(* PLC project SyntheticProject, CODESYS CODESYS V3.5 SP21 *)
(* stored: creationDateTime 2026-07-17T11:48:53, modificationDateTime 2026-07-17T11:48:53 *)

TYPE E_StationMode : (IDLE := 0, ACQUIRE := 10);
END_TYPE

TYPE E_MachineState : (OFF := 0);
END_TYPE

{attribute 'qualified_only'}
TYPE E_AlarmClass : (None := 0);
END_TYPE

TYPE ST_AxisConfig : STRUCT
  rMaxVel : REAL;  (* Max velocity *)
  rMaxAcc : REAL;  (* Max acceleration *)
  rMaxDec : REAL;  (* Max deceleration *)
  nAxisId : INT;  (* Axis identifier *)
  bInverted : BOOL;  (* Direction inverted *)
  tTimeout : TIME;  (* Motion timeout *)
END_STRUCT;
END_TYPE

TYPE ST_StationStats : STRUCT
  nTotalCycles : UDINT;  (* Total cycles run *)
  nFaultCount : DINT;  (* Fault count *)
  lrUptimeSec : LREAL;  (* Uptime in seconds *)
  rLastPos : REAL;  (* Last actual position *)
  sLastFault : STRING;  (* Last fault text *)
END_STRUCT;
END_TYPE

VAR_GLOBAL  (* GVL_Machine *)
  bMachineReady : BOOL;  (* Machine ready flag *)
  bEStop : BOOL;  (* Emergency stop active *)
  eMachineMode : E_MachineState;  (* Current machine state *)
  stAxisCfg : ST_AxisConfig;  (* Shared axis config *)
  nActiveStation : INT := 0;  (* Active station index *)
  rLineSpeed : REAL := 0.0;  (* Line speed *)
  lrProduced : LREAL := 0.0;  (* Produced count (long) *)
  tHeartbeat : TIME;  (* Heartbeat period *)
  sMachineName : STRING := 'LineA';  (* Machine name *)
END_VAR

VAR_GLOBAL CONSTANT  (* GVL_Config *)
  nMaxStations : INT := 24;  (* Max stations *)
  nBufferSize : UDINT := 256;  (* Buffer size *)
  rPi : REAL := 3.14159;  (* Pi constant *)
  lrGravity : LREAL := 9.80665;  (* Gravity constant *)
  tCycleTimeout : TIME := T#5S;  (* Default cycle timeout *)
  sVersion : STRING := '1.0.0';  (* Fixture version *)
END_VAR

VAR_GLOBAL RETAIN PERSISTENT  (* GVL_Persist *)
  nPowerCycles : UDINT := 0;  (* Power-cycle counter *)
  rTotalRuntime : LREAL := 0.0;  (* Accumulated runtime [h] *)
  nLastRecipeId : INT := 0;  (* Recipe restored on boot *)
END_VAR

FUNCTION_BLOCK FB_Debounce
  VAR_INPUT
    bIn : BOOL;  (* Raw input *)
    tDebounce : TIME := T#20MS;  (* Debounce time *)
  END_VAR
  VAR_OUTPUT
    bOut : BOOL;  (* Debounced output *)
  END_VAR
  VAR
    nState : INT := 0;  (* State machine *)
    bLast : BOOL;  (* Last raw sample *)
  END_VAR

          CASE nState OF
    0: // IDLE
        IF bIn <> bLast THEN
            nState := 10;
        END_IF
    10: // SETTLING
        bLast := bIn;
        bOut := bIn;
        nState := 0;
END_CASE
        
END_FUNCTION_BLOCK

FUNCTION_BLOCK FB_Delay
  VAR_INPUT
    bStart : BOOL;  (* Start the delay *)
    tDelay : TIME := T#1S;  (* Delay duration *)
  END_VAR
  VAR_OUTPUT
    bDone : BOOL;  (* Delay elapsed *)
  END_VAR
  VAR
    nState : INT := 0;  (* State machine *)
    tElapsed : TIME;  (* Accumulated time *)
  END_VAR

          CASE nState OF
    0: // IDLE
        bDone := FALSE;
        IF bStart THEN
            nState := 10;
        END_IF
    10: // TIMING
        bDone := TRUE;
        nState := 90;
    90: // DONE
        IF NOT bStart THEN
            nState := 0;
        END_IF
END_CASE
        
END_FUNCTION_BLOCK

FUNCTION_BLOCK FB_Station01
  VAR_INPUT
    bEnable : BOOL;  (* Enable this station *)
    bExecute : BOOL;  (* Trigger one work cycle *)
    bReset : BOOL;  (* Clear latched error *)
    nMode : INT := 0;  (* Operating mode selector *)
    rSetpoint : REAL := 0.0;  (* Target setpoint *)
    tTimeout : TIME := T#5S;  (* Watchdog timeout *)
    sLabel : STRING := 'station';  (* Human-readable label *)
    nStationId : DINT := 1;  (* Station identifier *)
  END_VAR
  VAR_OUTPUT
    bDone : BOOL;  (* Cycle finished *)
    bBusy : BOOL;  (* Cycle running *)
    bErr : BOOL;  (* Error latched *)
    nErrId : DINT := 0;  (* Active error code *)
    rActPos : REAL;  (* Actual position feedback *)
    nCycleCount : UDINT := 0;  (* Completed cycle counter *)
  END_VAR
  VAR
    nState : INT := 0;  (* State machine register *)
    fbSub : FB_Debounce;  (* Nested FB instance *)
    fbTimer : FB_Delay;  (* Nested FB instance *)
    anBuffer : ARRAY[0..9] OF INT;  (* Integer ring buffer *)
    arSamples : ARRAY[0..7] OF REAL;  (* Sample window *)
    lrAccum : LREAL := 0.0;  (* Long accumulator *)
    tElapsed : TIME;  (* Elapsed cycle time *)
    bInternal : BOOL;  (* Internal work flag *)
  END_VAR
  VAR CONSTANT
    nMaxRetries : INT := 3;  (* Retry limit *)
    rScale : REAL := 1.5;  (* Setpoint scale factor *)
  END_VAR

          // 01: main state machine — 0 IDLE / 10-20 WORK / 90 DONE / 99 ERROR
CASE nState OF
    0: // IDLE — wait for enable + execute
        bBusy := FALSE;
        bDone := FALSE;
        IF bEnable AND bExecute THEN
            nState := 10;
        END_IF

    10: // WORK: acquire
        bBusy := TRUE;
        nCycleCount := nCycleCount + 1;
        fbSub(bIn := bEnable);
        nState := 20;

    20: (* WORK: process the sample and compute position *)
        rActPos := rSetpoint * rScale;
        lrAccum := lrAccum + LREAL#TO_LREAL(rActPos);
        fbTimer(bStart := TRUE, tDelay := tTimeout);
        IF fbTimer.bDone THEN
            nState := 90;
        END_IF

    90: // DONE — publish result, return to idle
        bDone := TRUE;
        bBusy := FALSE;
        nState := 0;

    99: // ERROR — latch fault
        bErr := TRUE;
        nErrId := 16#8001;
        bBusy := FALSE;
END_CASE

// Global reset path
IF bReset THEN
    bErr := FALSE;
    nErrId := 0;
    nState := 0;
END_IF
        
END_FUNCTION_BLOCK

FUNCTION_BLOCK FB_Station02
  VAR_INPUT
    bEnable : BOOL;  (* Enable this station *)
    bExecute : BOOL;  (* Trigger one work cycle *)
    bReset : BOOL;  (* Clear latched error *)
    nMode : INT := 0;  (* Operating mode selector *)
    rSetpoint : REAL := 0.0;  (* Target setpoint *)
    tTimeout : TIME := T#5S;  (* Watchdog timeout *)
    sLabel : STRING := 'station';  (* Human-readable label *)
    nStationId : DINT := 2;  (* Station identifier *)
  END_VAR
  VAR_OUTPUT
    bDone : BOOL;  (* Cycle finished *)
    bBusy : BOOL;  (* Cycle running *)
    bErr : BOOL;  (* Error latched *)
    nErrId : DINT := 0;  (* Active error code *)
    rActPos : REAL;  (* Actual position feedback *)
    nCycleCount : UDINT := 0;  (* Completed cycle counter *)
  END_VAR
  VAR
    nState : INT := 0;  (* State machine register *)
    fbSub : FB_Debounce;  (* Nested FB instance *)
    fbTimer : FB_Delay;  (* Nested FB instance *)
    anBuffer : ARRAY[0..9] OF INT;  (* Integer ring buffer *)
    arSamples : ARRAY[0..7] OF REAL;  (* Sample window *)
    lrAccum : LREAL := 0.0;  (* Long accumulator *)
    tElapsed : TIME;  (* Elapsed cycle time *)
    bInternal : BOOL;  (* Internal work flag *)
  END_VAR
  VAR CONSTANT
    nMaxRetries : INT := 3;  (* Retry limit *)
    rScale : REAL := 1.5;  (* Setpoint scale factor *)
  END_VAR

          // 02: main state machine — 0 IDLE / 10-20 WORK / 90 DONE / 99 ERROR
CASE nState OF
    0: // IDLE — wait for enable + execute
        bBusy := FALSE;
        bDone := FALSE;
        IF bEnable AND bExecute THEN
            nState := 10;
        END_IF

    10: // WORK: acquire
        bBusy := TRUE;
        nCycleCount := nCycleCount + 1;
        fbSub(bIn := bEnable);
        nState := 20;

    20: (* WORK: process the sample and compute position *)
        rActPos := rSetpoint * rScale;
        lrAccum := lrAccum + LREAL#TO_LREAL(rActPos);
        fbTimer(bStart := TRUE, tDelay := tTimeout);
        IF fbTimer.bDone THEN
            nState := 90;
        END_IF

    90: // DONE — publish result, return to idle
        bDone := TRUE;
        bBusy := FALSE;
        nState := 0;

    99: // ERROR — latch fault
        bErr := TRUE;
        nErrId := 16#8001;
        bBusy := FALSE;
END_CASE

// Global reset path
IF bReset THEN
    bErr := FALSE;
    nErrId := 0;
    nState := 0;
END_IF
        
END_FUNCTION_BLOCK

FUNCTION_BLOCK FB_Station03
  VAR_INPUT
    bEnable : BOOL;  (* Enable this station *)
    bExecute : BOOL;  (* Trigger one work cycle *)
    bReset : BOOL;  (* Clear latched error *)
    nMode : INT := 0;  (* Operating mode selector *)
    rSetpoint : REAL := 0.0;  (* Target setpoint *)
    tTimeout : TIME := T#5S;  (* Watchdog timeout *)
    sLabel : STRING := 'station';  (* Human-readable label *)
    nStationId : DINT := 3;  (* Station identifier *)
  END_VAR
  VAR_OUTPUT
    bDone : BOOL;  (* Cycle finished *)
    bBusy : BOOL;  (* Cycle running *)
    bErr : BOOL;  (* Error latched *)
    nErrId : DINT := 0;  (* Active error code *)
    rActPos : REAL;  (* Actual position feedback *)
    nCycleCount : UDINT := 0;  (* Completed cycle counter *)
  END_VAR
  VAR
    nState : INT := 0;  (* State machine register *)
    fbSub : FB_Debounce;  (* Nested FB instance *)
    fbTimer : FB_Delay;  (* Nested FB instance *)
    anBuffer : ARRAY[0..9] OF INT;  (* Integer ring buffer *)
    arSamples : ARRAY[0..7] OF REAL;  (* Sample window *)
    lrAccum : LREAL := 0.0;  (* Long accumulator *)
    tElapsed : TIME;  (* Elapsed cycle time *)
    bInternal : BOOL;  (* Internal work flag *)
  END_VAR
  VAR CONSTANT
    nMaxRetries : INT := 3;  (* Retry limit *)
    rScale : REAL := 1.5;  (* Setpoint scale factor *)
  END_VAR

          // 03: main state machine — 0 IDLE / 10-20 WORK / 90 DONE / 99 ERROR
CASE nState OF
    0: // IDLE — wait for enable + execute
        bBusy := FALSE;
        bDone := FALSE;
        IF bEnable AND bExecute THEN
            nState := 10;
        END_IF

    10: // WORK: acquire
        bBusy := TRUE;
        nCycleCount := nCycleCount + 1;
        fbSub(bIn := bEnable);
        nState := 20;

    20: (* WORK: process the sample and compute position *)
        rActPos := rSetpoint * rScale;
        lrAccum := lrAccum + LREAL#TO_LREAL(rActPos);
        fbTimer(bStart := TRUE, tDelay := tTimeout);
        IF fbTimer.bDone THEN
            nState := 90;
        END_IF

    90: // DONE — publish result, return to idle
        bDone := TRUE;
        bBusy := FALSE;
        nState := 0;

    99: // ERROR — latch fault
        bErr := TRUE;
        nErrId := 16#8001;
        bBusy := FALSE;
END_CASE

// Global reset path
IF bReset THEN
    bErr := FALSE;
    nErrId := 0;
    nState := 0;
END_IF
        
END_FUNCTION_BLOCK

FUNCTION_BLOCK FB_Station04
  VAR_INPUT
    bEnable : BOOL;  (* Enable this station *)
    bExecute : BOOL;  (* Trigger one work cycle *)
    bReset : BOOL;  (* Clear latched error *)
    nMode : INT := 0;  (* Operating mode selector *)
    rSetpoint : REAL := 0.0;  (* Target setpoint *)
    tTimeout : TIME := T#5S;  (* Watchdog timeout *)
    sLabel : STRING := 'station';  (* Human-readable label *)
    nStationId : DINT := 4;  (* Station identifier *)
  END_VAR
  VAR_OUTPUT
    bDone : BOOL;  (* Cycle finished *)
    bBusy : BOOL;  (* Cycle running *)
    bErr : BOOL;  (* Error latched *)
    nErrId : DINT := 0;  (* Active error code *)
    rActPos : REAL;  (* Actual position feedback *)
    nCycleCount : UDINT := 0;  (* Completed cycle counter *)
  END_VAR
  VAR
    nState : INT := 0;  (* State machine register *)
    fbSub : FB_Debounce;  (* Nested FB instance *)
    fbTimer : FB_Delay;  (* Nested FB instance *)
    anBuffer : ARRAY[0..9] OF INT;  (* Integer ring buffer *)
    arSamples : ARRAY[0..7] OF REAL;  (* Sample window *)
    lrAccum : LREAL := 0.0;  (* Long accumulator *)
    tElapsed : TIME;  (* Elapsed cycle time *)
    bInternal : BOOL;  (* Internal work flag *)
  END_VAR
  VAR CONSTANT
    nMaxRetries : INT := 3;  (* Retry limit *)
    rScale : REAL := 1.5;  (* Setpoint scale factor *)
  END_VAR

          // 04: main state machine — 0 IDLE / 10-20 WORK / 90 DONE / 99 ERROR
CASE nState OF
    0: // IDLE — wait for enable + execute
        bBusy := FALSE;
        bDone := FALSE;
        IF bEnable AND bExecute THEN
            nState := 10;
        END_IF

    10: // WORK: acquire
        bBusy := TRUE;
        nCycleCount := nCycleCount + 1;
        fbSub(bIn := bEnable);
        nState := 20;

    20: (* WORK: process the sample and compute position *)
        rActPos := rSetpoint * rScale;
        lrAccum := lrAccum + LREAL#TO_LREAL(rActPos);
        fbTimer(bStart := TRUE, tDelay := tTimeout);
        IF fbTimer.bDone THEN
            nState := 90;
        END_IF

    90: // DONE — publish result, return to idle
        bDone := TRUE;
        bBusy := FALSE;
        nState := 0;

    99: // ERROR — latch fault
        bErr := TRUE;
        nErrId := 16#8001;
        bBusy := FALSE;
END_CASE

// Global reset path
IF bReset THEN
    bErr := FALSE;
    nErrId := 0;
    nState := 0;
END_IF
        
END_FUNCTION_BLOCK

FUNCTION_BLOCK FB_Station05
  VAR_INPUT
    bEnable : BOOL;  (* Enable this station *)
    bExecute : BOOL;  (* Trigger one work cycle *)
    bReset : BOOL;  (* Clear latched error *)
    nMode : INT := 0;  (* Operating mode selector *)
    rSetpoint : REAL := 0.0;  (* Target setpoint *)
    tTimeout : TIME := T#5S;  (* Watchdog timeout *)
    sLabel : STRING := 'station';  (* Human-readable label *)
    nStationId : DINT := 5;  (* Station identifier *)
  END_VAR
  VAR_OUTPUT
    bDone : BOOL;  (* Cycle finished *)
    bBusy : BOOL;  (* Cycle running *)
    bErr : BOOL;  (* Error latched *)
    nErrId : DINT := 0;  (* Active error code *)
    rActPos : REAL;  (* Actual position feedback *)
    nCycleCount : UDINT := 0;  (* Completed cycle counter *)
  END_VAR
  VAR
    nState : INT := 0;  (* State machine register *)
    fbSub : FB_Debounce;  (* Nested FB instance *)
    fbTimer : FB_Delay;  (* Nested FB instance *)
    anBuffer : ARRAY[0..9] OF INT;  (* Integer ring buffer *)
    arSamples : ARRAY[0..7] OF REAL;  (* Sample window *)
    lrAccum : LREAL := 0.0;  (* Long accumulator *)
    tElapsed : TIME;  (* Elapsed cycle time *)
    bInternal : BOOL;  (* Internal work flag *)
  END_VAR
  VAR CONSTANT
    nMaxRetries : INT := 3;  (* Retry limit *)
    rScale : REAL := 1.5;  (* Setpoint scale factor *)
  END_VAR

          // 05: main state machine — 0 IDLE / 10-20 WORK / 90 DONE / 99 ERROR
CASE nState OF
    0: // IDLE — wait for enable + execute
        bBusy := FALSE;
        bDone := FALSE;
        IF bEnable AND bExecute THEN
            nState := 10;
        END_IF

    10: // WORK: acquire
        bBusy := TRUE;
        nCycleCount := nCycleCount + 1;
        fbSub(bIn := bEnable);
        nState := 20;

    20: (* WORK: process the sample and compute position *)
        rActPos := rSetpoint * rScale;
        lrAccum := lrAccum + LREAL#TO_LREAL(rActPos);
        fbTimer(bStart := TRUE, tDelay := tTimeout);
        IF fbTimer.bDone THEN
            nState := 90;
        END_IF

    90: // DONE — publish result, return to idle
        bDone := TRUE;
        bBusy := FALSE;
        nState := 0;

    99: // ERROR — latch fault
        bErr := TRUE;
        nErrId := 16#8001;
        bBusy := FALSE;
END_CASE

// Global reset path
IF bReset THEN
    bErr := FALSE;
    nErrId := 0;
    nState := 0;
END_IF
        
END_FUNCTION_BLOCK

FUNCTION_BLOCK FB_Station06
  VAR_INPUT
    bEnable : BOOL;  (* Enable this station *)
    bExecute : BOOL;  (* Trigger one work cycle *)
    bReset : BOOL;  (* Clear latched error *)
    nMode : INT := 0;  (* Operating mode selector *)
    rSetpoint : REAL := 0.0;  (* Target setpoint *)
    tTimeout : TIME := T#5S;  (* Watchdog timeout *)
    sLabel : STRING := 'station';  (* Human-readable label *)
    nStationId : DINT := 6;  (* Station identifier *)
  END_VAR
  VAR_OUTPUT
    bDone : BOOL;  (* Cycle finished *)
    bBusy : BOOL;  (* Cycle running *)
    bErr : BOOL;  (* Error latched *)
    nErrId : DINT := 0;  (* Active error code *)
    rActPos : REAL;  (* Actual position feedback *)
    nCycleCount : UDINT := 0;  (* Completed cycle counter *)
  END_VAR
  VAR
    nState : INT := 0;  (* State machine register *)
    fbSub : FB_Debounce;  (* Nested FB instance *)
    fbTimer : FB_Delay;  (* Nested FB instance *)
    anBuffer : ARRAY[0..9] OF INT;  (* Integer ring buffer *)
    arSamples : ARRAY[0..7] OF REAL;  (* Sample window *)
    lrAccum : LREAL := 0.0;  (* Long accumulator *)
    tElapsed : TIME;  (* Elapsed cycle time *)
    bInternal : BOOL;  (* Internal work flag *)
  END_VAR
  VAR CONSTANT
    nMaxRetries : INT := 3;  (* Retry limit *)
    rScale : REAL := 1.5;  (* Setpoint scale factor *)
  END_VAR

          // 06: main state machine — 0 IDLE / 10-20 WORK / 90 DONE / 99 ERROR
CASE nState OF
    0: // IDLE — wait for enable + execute
        bBusy := FALSE;
        bDone := FALSE;
        IF bEnable AND bExecute THEN
            nState := 10;
        END_IF

    10: // WORK: acquire
        bBusy := TRUE;
        nCycleCount := nCycleCount + 1;
        fbSub(bIn := bEnable);
        nState := 20;

    20: (* WORK: process the sample and compute position *)
        rActPos := rSetpoint * rScale;
        lrAccum := lrAccum + LREAL#TO_LREAL(rActPos);
        fbTimer(bStart := TRUE, tDelay := tTimeout);
        IF fbTimer.bDone THEN
            nState := 90;
        END_IF

    90: // DONE — publish result, return to idle
        bDone := TRUE;
        bBusy := FALSE;
        nState := 0;

    99: // ERROR — latch fault
        bErr := TRUE;
        nErrId := 16#8001;
        bBusy := FALSE;
END_CASE

// Global reset path
IF bReset THEN
    bErr := FALSE;
    nErrId := 0;
    nState := 0;
END_IF
        
END_FUNCTION_BLOCK

FUNCTION_BLOCK FB_Station07
  VAR_INPUT
    bEnable : BOOL;  (* Enable this station *)
    bExecute : BOOL;  (* Trigger one work cycle *)
    bReset : BOOL;  (* Clear latched error *)
    nMode : INT := 0;  (* Operating mode selector *)
    rSetpoint : REAL := 0.0;  (* Target setpoint *)
    tTimeout : TIME := T#5S;  (* Watchdog timeout *)
    sLabel : STRING := 'station';  (* Human-readable label *)
    nStationId : DINT := 7;  (* Station identifier *)
  END_VAR
  VAR_OUTPUT
    bDone : BOOL;  (* Cycle finished *)
    bBusy : BOOL;  (* Cycle running *)
    bErr : BOOL;  (* Error latched *)
    nErrId : DINT := 0;  (* Active error code *)
    rActPos : REAL;  (* Actual position feedback *)
    nCycleCount : UDINT := 0;  (* Completed cycle counter *)
  END_VAR
  VAR
    nState : INT := 0;  (* State machine register *)
    fbSub : FB_Debounce;  (* Nested FB instance *)
    fbTimer : FB_Delay;  (* Nested FB instance *)
    anBuffer : ARRAY[0..9] OF INT;  (* Integer ring buffer *)
    arSamples : ARRAY[0..7] OF REAL;  (* Sample window *)
    lrAccum : LREAL := 0.0;  (* Long accumulator *)
    tElapsed : TIME;  (* Elapsed cycle time *)
    bInternal : BOOL;  (* Internal work flag *)
  END_VAR
  VAR CONSTANT
    nMaxRetries : INT := 3;  (* Retry limit *)
    rScale : REAL := 1.5;  (* Setpoint scale factor *)
  END_VAR

          // 07: main state machine — 0 IDLE / 10-20 WORK / 90 DONE / 99 ERROR
CASE nState OF
    0: // IDLE — wait for enable + execute
        bBusy := FALSE;
        bDone := FALSE;
        IF bEnable AND bExecute THEN
            nState := 10;
        END_IF

    10: // WORK: acquire
        bBusy := TRUE;
        nCycleCount := nCycleCount + 1;
        fbSub(bIn := bEnable);
        nState := 20;

    20: (* WORK: process the sample and compute position *)
        rActPos := rSetpoint * rScale;
        lrAccum := lrAccum + LREAL#TO_LREAL(rActPos);
        fbTimer(bStart := TRUE, tDelay := tTimeout);
        IF fbTimer.bDone THEN
            nState := 90;
        END_IF

    90: // DONE — publish result, return to idle
        bDone := TRUE;
        bBusy := FALSE;
        nState := 0;

    99: // ERROR — latch fault
        bErr := TRUE;
        nErrId := 16#8001;
        bBusy := FALSE;
END_CASE

// Global reset path
IF bReset THEN
    bErr := FALSE;
    nErrId := 0;
    nState := 0;
END_IF
        
END_FUNCTION_BLOCK

FUNCTION_BLOCK FB_Station08
  VAR_INPUT
    bEnable : BOOL;  (* Enable this station *)
    bExecute : BOOL;  (* Trigger one work cycle *)
    bReset : BOOL;  (* Clear latched error *)
    nMode : INT := 0;  (* Operating mode selector *)
    rSetpoint : REAL := 0.0;  (* Target setpoint *)
    tTimeout : TIME := T#5S;  (* Watchdog timeout *)
    sLabel : STRING := 'station';  (* Human-readable label *)
    nStationId : DINT := 8;  (* Station identifier *)
  END_VAR
  VAR_OUTPUT
    bDone : BOOL;  (* Cycle finished *)
    bBusy : BOOL;  (* Cycle running *)
    bErr : BOOL;  (* Error latched *)
    nErrId : DINT := 0;  (* Active error code *)
    rActPos : REAL;  (* Actual position feedback *)
    nCycleCount : UDINT := 0;  (* Completed cycle counter *)
  END_VAR
  VAR
    nState : INT := 0;  (* State machine register *)
    fbSub : FB_Debounce;  (* Nested FB instance *)
    fbTimer : FB_Delay;  (* Nested FB instance *)
    anBuffer : ARRAY[0..9] OF INT;  (* Integer ring buffer *)
    arSamples : ARRAY[0..7] OF REAL;  (* Sample window *)
    lrAccum : LREAL := 0.0;  (* Long accumulator *)
    tElapsed : TIME;  (* Elapsed cycle time *)
    bInternal : BOOL;  (* Internal work flag *)
  END_VAR
  VAR CONSTANT
    nMaxRetries : INT := 3;  (* Retry limit *)
    rScale : REAL := 1.5;  (* Setpoint scale factor *)
  END_VAR

          // 08: main state machine — 0 IDLE / 10-20 WORK / 90 DONE / 99 ERROR
CASE nState OF
    0: // IDLE — wait for enable + execute
        bBusy := FALSE;
        bDone := FALSE;
        IF bEnable AND bExecute THEN
            nState := 10;
        END_IF

    10: // WORK: acquire
        bBusy := TRUE;
        nCycleCount := nCycleCount + 1;
        fbSub(bIn := bEnable);
        nState := 20;

    20: (* WORK: process the sample and compute position *)
        rActPos := rSetpoint * rScale;
        lrAccum := lrAccum + LREAL#TO_LREAL(rActPos);
        fbTimer(bStart := TRUE, tDelay := tTimeout);
        IF fbTimer.bDone THEN
            nState := 90;
        END_IF

    90: // DONE — publish result, return to idle
        bDone := TRUE;
        bBusy := FALSE;
        nState := 0;

    99: // ERROR — latch fault
        bErr := TRUE;
        nErrId := 16#8001;
        bBusy := FALSE;
END_CASE

// Global reset path
IF bReset THEN
    bErr := FALSE;
    nErrId := 0;
    nState := 0;
END_IF
        
END_FUNCTION_BLOCK

FUNCTION_BLOCK FB_Station09
  VAR_INPUT
    bEnable : BOOL;  (* Enable this station *)
    bExecute : BOOL;  (* Trigger one work cycle *)
    bReset : BOOL;  (* Clear latched error *)
    nMode : INT := 0;  (* Operating mode selector *)
    rSetpoint : REAL := 0.0;  (* Target setpoint *)
    tTimeout : TIME := T#5S;  (* Watchdog timeout *)
    sLabel : STRING := 'station';  (* Human-readable label *)
    nStationId : DINT := 9;  (* Station identifier *)
  END_VAR
  VAR_OUTPUT
    bDone : BOOL;  (* Cycle finished *)
    bBusy : BOOL;  (* Cycle running *)
    bErr : BOOL;  (* Error latched *)
    nErrId : DINT := 0;  (* Active error code *)
    rActPos : REAL;  (* Actual position feedback *)
    nCycleCount : UDINT := 0;  (* Completed cycle counter *)
  END_VAR
  VAR
    nState : INT := 0;  (* State machine register *)
    fbSub : FB_Debounce;  (* Nested FB instance *)
    fbTimer : FB_Delay;  (* Nested FB instance *)
    anBuffer : ARRAY[0..9] OF INT;  (* Integer ring buffer *)
    arSamples : ARRAY[0..7] OF REAL;  (* Sample window *)
    lrAccum : LREAL := 0.0;  (* Long accumulator *)
    tElapsed : TIME;  (* Elapsed cycle time *)
    bInternal : BOOL;  (* Internal work flag *)
  END_VAR
  VAR CONSTANT
    nMaxRetries : INT := 3;  (* Retry limit *)
    rScale : REAL := 1.5;  (* Setpoint scale factor *)
  END_VAR

          // 09: main state machine — 0 IDLE / 10-20 WORK / 90 DONE / 99 ERROR
CASE nState OF
    0: // IDLE — wait for enable + execute
        bBusy := FALSE;
        bDone := FALSE;
        IF bEnable AND bExecute THEN
            nState := 10;
        END_IF

    10: // WORK: acquire
        bBusy := TRUE;
        nCycleCount := nCycleCount + 1;
        fbSub(bIn := bEnable);
        nState := 20;

    20: (* WORK: process the sample and compute position *)
        rActPos := rSetpoint * rScale;
        lrAccum := lrAccum + LREAL#TO_LREAL(rActPos);
        fbTimer(bStart := TRUE, tDelay := tTimeout);
        IF fbTimer.bDone THEN
            nState := 90;
        END_IF

    90: // DONE — publish result, return to idle
        bDone := TRUE;
        bBusy := FALSE;
        nState := 0;

    99: // ERROR — latch fault
        bErr := TRUE;
        nErrId := 16#8001;
        bBusy := FALSE;
END_CASE

// Global reset path
IF bReset THEN
    bErr := FALSE;
    nErrId := 0;
    nState := 0;
END_IF
        
END_FUNCTION_BLOCK

FUNCTION_BLOCK FB_Station10
  VAR_INPUT
    bEnable : BOOL;  (* Enable this station *)
    bExecute : BOOL;  (* Trigger one work cycle *)
    bReset : BOOL;  (* Clear latched error *)
    nMode : INT := 0;  (* Operating mode selector *)
    rSetpoint : REAL := 0.0;  (* Target setpoint *)
    tTimeout : TIME := T#5S;  (* Watchdog timeout *)
    sLabel : STRING := 'station';  (* Human-readable label *)
    nStationId : DINT := 10;  (* Station identifier *)
  END_VAR
  VAR_OUTPUT
    bDone : BOOL;  (* Cycle finished *)
    bBusy : BOOL;  (* Cycle running *)
    bErr : BOOL;  (* Error latched *)
    nErrId : DINT := 0;  (* Active error code *)
    rActPos : REAL;  (* Actual position feedback *)
    nCycleCount : UDINT := 0;  (* Completed cycle counter *)
  END_VAR
  VAR
    nState : INT := 0;  (* State machine register *)
    fbSub : FB_Debounce;  (* Nested FB instance *)
    fbTimer : FB_Delay;  (* Nested FB instance *)
    anBuffer : ARRAY[0..9] OF INT;  (* Integer ring buffer *)
    arSamples : ARRAY[0..7] OF REAL;  (* Sample window *)
    lrAccum : LREAL := 0.0;  (* Long accumulator *)
    tElapsed : TIME;  (* Elapsed cycle time *)
    bInternal : BOOL;  (* Internal work flag *)
  END_VAR
  VAR CONSTANT
    nMaxRetries : INT := 3;  (* Retry limit *)
    rScale : REAL := 1.5;  (* Setpoint scale factor *)
  END_VAR

          // 10: main state machine — 0 IDLE / 10-20 WORK / 90 DONE / 99 ERROR
CASE nState OF
    0: // IDLE — wait for enable + execute
        bBusy := FALSE;
        bDone := FALSE;
        IF bEnable AND bExecute THEN
            nState := 10;
        END_IF

    10: // WORK: acquire
        bBusy := TRUE;
        nCycleCount := nCycleCount + 1;
        fbSub(bIn := bEnable);
        nState := 20;

    20: (* WORK: process the sample and compute position *)
        rActPos := rSetpoint * rScale;
        lrAccum := lrAccum + LREAL#TO_LREAL(rActPos);
        fbTimer(bStart := TRUE, tDelay := tTimeout);
        IF fbTimer.bDone THEN
            nState := 90;
        END_IF

    90: // DONE — publish result, return to idle
        bDone := TRUE;
        bBusy := FALSE;
        nState := 0;

    99: // ERROR — latch fault
        bErr := TRUE;
        nErrId := 16#8001;
        bBusy := FALSE;
END_CASE

// Global reset path
IF bReset THEN
    bErr := FALSE;
    nErrId := 0;
    nState := 0;
END_IF
        
END_FUNCTION_BLOCK

FUNCTION_BLOCK FB_Station11
  VAR_INPUT
    bEnable : BOOL;  (* Enable this station *)
    bExecute : BOOL;  (* Trigger one work cycle *)
    bReset : BOOL;  (* Clear latched error *)
    nMode : INT := 0;  (* Operating mode selector *)
    rSetpoint : REAL := 0.0;  (* Target setpoint *)
    tTimeout : TIME := T#5S;  (* Watchdog timeout *)
    sLabel : STRING := 'station';  (* Human-readable label *)
    nStationId : DINT := 11;  (* Station identifier *)
  END_VAR
  VAR_OUTPUT
    bDone : BOOL;  (* Cycle finished *)
    bBusy : BOOL;  (* Cycle running *)
    bErr : BOOL;  (* Error latched *)
    nErrId : DINT := 0;  (* Active error code *)
    rActPos : REAL;  (* Actual position feedback *)
    nCycleCount : UDINT := 0;  (* Completed cycle counter *)
  END_VAR
  VAR
    nState : INT := 0;  (* State machine register *)
    fbSub : FB_Debounce;  (* Nested FB instance *)
    fbTimer : FB_Delay;  (* Nested FB instance *)
    anBuffer : ARRAY[0..9] OF INT;  (* Integer ring buffer *)
    arSamples : ARRAY[0..7] OF REAL;  (* Sample window *)
    lrAccum : LREAL := 0.0;  (* Long accumulator *)
    tElapsed : TIME;  (* Elapsed cycle time *)
    bInternal : BOOL;  (* Internal work flag *)
  END_VAR
  VAR CONSTANT
    nMaxRetries : INT := 3;  (* Retry limit *)
    rScale : REAL := 1.5;  (* Setpoint scale factor *)
  END_VAR

          // 11: main state machine — 0 IDLE / 10-20 WORK / 90 DONE / 99 ERROR
CASE nState OF
    0: // IDLE — wait for enable + execute
        bBusy := FALSE;
        bDone := FALSE;
        IF bEnable AND bExecute THEN
            nState := 10;
        END_IF

    10: // WORK: acquire
        bBusy := TRUE;
        nCycleCount := nCycleCount + 1;
        fbSub(bIn := bEnable);
        nState := 20;

    20: (* WORK: process the sample and compute position *)
        rActPos := rSetpoint * rScale;
        lrAccum := lrAccum + LREAL#TO_LREAL(rActPos);
        fbTimer(bStart := TRUE, tDelay := tTimeout);
        IF fbTimer.bDone THEN
            nState := 90;
        END_IF

    90: // DONE — publish result, return to idle
        bDone := TRUE;
        bBusy := FALSE;
        nState := 0;

    99: // ERROR — latch fault
        bErr := TRUE;
        nErrId := 16#8001;
        bBusy := FALSE;
END_CASE

// Global reset path
IF bReset THEN
    bErr := FALSE;
    nErrId := 0;
    nState := 0;
END_IF
        
END_FUNCTION_BLOCK

FUNCTION_BLOCK FB_Station12
  VAR_INPUT
    bEnable : BOOL;  (* Enable this station *)
    bExecute : BOOL;  (* Trigger one work cycle *)
    bReset : BOOL;  (* Clear latched error *)
    nMode : INT := 0;  (* Operating mode selector *)
    rSetpoint : REAL := 0.0;  (* Target setpoint *)
    tTimeout : TIME := T#5S;  (* Watchdog timeout *)
    sLabel : STRING := 'station';  (* Human-readable label *)
    nStationId : DINT := 12;  (* Station identifier *)
  END_VAR
  VAR_OUTPUT
    bDone : BOOL;  (* Cycle finished *)
    bBusy : BOOL;  (* Cycle running *)
    bErr : BOOL;  (* Error latched *)
    nErrId : DINT := 0;  (* Active error code *)
    rActPos : REAL;  (* Actual position feedback *)
    nCycleCount : UDINT := 0;  (* Completed cycle counter *)
  END_VAR
  VAR
    nState : INT := 0;  (* State machine register *)
    fbSub : FB_Debounce;  (* Nested FB instance *)
    fbTimer : FB_Delay;  (* Nested FB instance *)
    anBuffer : ARRAY[0..9] OF INT;  (* Integer ring buffer *)
    arSamples : ARRAY[0..7] OF REAL;  (* Sample window *)
    lrAccum : LREAL := 0.0;  (* Long accumulator *)
    tElapsed : TIME;  (* Elapsed cycle time *)
    bInternal : BOOL;  (* Internal work flag *)
  END_VAR
  VAR CONSTANT
    nMaxRetries : INT := 3;  (* Retry limit *)
    rScale : REAL := 1.5;  (* Setpoint scale factor *)
  END_VAR

          // 12: main state machine — 0 IDLE / 10-20 WORK / 90 DONE / 99 ERROR
CASE nState OF
    0: // IDLE — wait for enable + execute
        bBusy := FALSE;
        bDone := FALSE;
        IF bEnable AND bExecute THEN
            nState := 10;
        END_IF

    10: // WORK: acquire
        bBusy := TRUE;
        nCycleCount := nCycleCount + 1;
        fbSub(bIn := bEnable);
        nState := 20;

    20: (* WORK: process the sample and compute position *)
        rActPos := rSetpoint * rScale;
        lrAccum := lrAccum + LREAL#TO_LREAL(rActPos);
        fbTimer(bStart := TRUE, tDelay := tTimeout);
        IF fbTimer.bDone THEN
            nState := 90;
        END_IF

    90: // DONE — publish result, return to idle
        bDone := TRUE;
        bBusy := FALSE;
        nState := 0;

    99: // ERROR — latch fault
        bErr := TRUE;
        nErrId := 16#8001;
        bBusy := FALSE;
END_CASE

// Global reset path
IF bReset THEN
    bErr := FALSE;
    nErrId := 0;
    nState := 0;
END_IF
        
END_FUNCTION_BLOCK

FUNCTION_BLOCK FB_Station13
  VAR_INPUT
    bEnable : BOOL;  (* Enable this station *)
    bExecute : BOOL;  (* Trigger one work cycle *)
    bReset : BOOL;  (* Clear latched error *)
    nMode : INT := 0;  (* Operating mode selector *)
    rSetpoint : REAL := 0.0;  (* Target setpoint *)
    tTimeout : TIME := T#5S;  (* Watchdog timeout *)
    sLabel : STRING := 'station';  (* Human-readable label *)
    nStationId : DINT := 13;  (* Station identifier *)
  END_VAR
  VAR_OUTPUT
    bDone : BOOL;  (* Cycle finished *)
    bBusy : BOOL;  (* Cycle running *)
    bErr : BOOL;  (* Error latched *)
    nErrId : DINT := 0;  (* Active error code *)
    rActPos : REAL;  (* Actual position feedback *)
    nCycleCount : UDINT := 0;  (* Completed cycle counter *)
  END_VAR
  VAR
    nState : INT := 0;  (* State machine register *)
    fbSub : FB_Debounce;  (* Nested FB instance *)
    fbTimer : FB_Delay;  (* Nested FB instance *)
    anBuffer : ARRAY[0..9] OF INT;  (* Integer ring buffer *)
    arSamples : ARRAY[0..7] OF REAL;  (* Sample window *)
    lrAccum : LREAL := 0.0;  (* Long accumulator *)
    tElapsed : TIME;  (* Elapsed cycle time *)
    bInternal : BOOL;  (* Internal work flag *)
  END_VAR
  VAR CONSTANT
    nMaxRetries : INT := 3;  (* Retry limit *)
    rScale : REAL := 1.5;  (* Setpoint scale factor *)
  END_VAR

          // 13: main state machine — 0 IDLE / 10-20 WORK / 90 DONE / 99 ERROR
CASE nState OF
    0: // IDLE — wait for enable + execute
        bBusy := FALSE;
        bDone := FALSE;
        IF bEnable AND bExecute THEN
            nState := 10;
        END_IF

    10: // WORK: acquire
        bBusy := TRUE;
        nCycleCount := nCycleCount + 1;
        fbSub(bIn := bEnable);
        nState := 20;

    20: (* WORK: process the sample and compute position *)
        rActPos := rSetpoint * rScale;
        lrAccum := lrAccum + LREAL#TO_LREAL(rActPos);
        fbTimer(bStart := TRUE, tDelay := tTimeout);
        IF fbTimer.bDone THEN
            nState := 90;
        END_IF

    90: // DONE — publish result, return to idle
        bDone := TRUE;
        bBusy := FALSE;
        nState := 0;

    99: // ERROR — latch fault
        bErr := TRUE;
        nErrId := 16#8001;
        bBusy := FALSE;
END_CASE

// Global reset path
IF bReset THEN
    bErr := FALSE;
    nErrId := 0;
    nState := 0;
END_IF
        
END_FUNCTION_BLOCK

FUNCTION_BLOCK FB_Station14
  VAR_INPUT
    bEnable : BOOL;  (* Enable this station *)
    bExecute : BOOL;  (* Trigger one work cycle *)
    bReset : BOOL;  (* Clear latched error *)
    nMode : INT := 0;  (* Operating mode selector *)
    rSetpoint : REAL := 0.0;  (* Target setpoint *)
    tTimeout : TIME := T#5S;  (* Watchdog timeout *)
    sLabel : STRING := 'station';  (* Human-readable label *)
    nStationId : DINT := 14;  (* Station identifier *)
  END_VAR
  VAR_OUTPUT
    bDone : BOOL;  (* Cycle finished *)
    bBusy : BOOL;  (* Cycle running *)
    bErr : BOOL;  (* Error latched *)
    nErrId : DINT := 0;  (* Active error code *)
    rActPos : REAL;  (* Actual position feedback *)
    nCycleCount : UDINT := 0;  (* Completed cycle counter *)
  END_VAR
  VAR
    nState : INT := 0;  (* State machine register *)
    fbSub : FB_Debounce;  (* Nested FB instance *)
    fbTimer : FB_Delay;  (* Nested FB instance *)
    anBuffer : ARRAY[0..9] OF INT;  (* Integer ring buffer *)
    arSamples : ARRAY[0..7] OF REAL;  (* Sample window *)
    lrAccum : LREAL := 0.0;  (* Long accumulator *)
    tElapsed : TIME;  (* Elapsed cycle time *)
    bInternal : BOOL;  (* Internal work flag *)
  END_VAR
  VAR CONSTANT
    nMaxRetries : INT := 3;  (* Retry limit *)
    rScale : REAL := 1.5;  (* Setpoint scale factor *)
  END_VAR

          // 14: main state machine — 0 IDLE / 10-20 WORK / 90 DONE / 99 ERROR
CASE nState OF
    0: // IDLE — wait for enable + execute
        bBusy := FALSE;
        bDone := FALSE;
        IF bEnable AND bExecute THEN
            nState := 10;
        END_IF

    10: // WORK: acquire
        bBusy := TRUE;
        nCycleCount := nCycleCount + 1;
        fbSub(bIn := bEnable);
        nState := 20;

    20: (* WORK: process the sample and compute position *)
        rActPos := rSetpoint * rScale;
        lrAccum := lrAccum + LREAL#TO_LREAL(rActPos);
        fbTimer(bStart := TRUE, tDelay := tTimeout);
        IF fbTimer.bDone THEN
            nState := 90;
        END_IF

    90: // DONE — publish result, return to idle
        bDone := TRUE;
        bBusy := FALSE;
        nState := 0;

    99: // ERROR — latch fault
        bErr := TRUE;
        nErrId := 16#8001;
        bBusy := FALSE;
END_CASE

// Global reset path
IF bReset THEN
    bErr := FALSE;
    nErrId := 0;
    nState := 0;
END_IF
        
END_FUNCTION_BLOCK

FUNCTION_BLOCK FB_Station15
  VAR_INPUT
    bEnable : BOOL;  (* Enable this station *)
    bExecute : BOOL;  (* Trigger one work cycle *)
    bReset : BOOL;  (* Clear latched error *)
    nMode : INT := 0;  (* Operating mode selector *)
    rSetpoint : REAL := 0.0;  (* Target setpoint *)
    tTimeout : TIME := T#5S;  (* Watchdog timeout *)
    sLabel : STRING := 'station';  (* Human-readable label *)
    nStationId : DINT := 15;  (* Station identifier *)
  END_VAR
  VAR_OUTPUT
    bDone : BOOL;  (* Cycle finished *)
    bBusy : BOOL;  (* Cycle running *)
    bErr : BOOL;  (* Error latched *)
    nErrId : DINT := 0;  (* Active error code *)
    rActPos : REAL;  (* Actual position feedback *)
    nCycleCount : UDINT := 0;  (* Completed cycle counter *)
  END_VAR
  VAR
    nState : INT := 0;  (* State machine register *)
    fbSub : FB_Debounce;  (* Nested FB instance *)
    fbTimer : FB_Delay;  (* Nested FB instance *)
    anBuffer : ARRAY[0..9] OF INT;  (* Integer ring buffer *)
    arSamples : ARRAY[0..7] OF REAL;  (* Sample window *)
    lrAccum : LREAL := 0.0;  (* Long accumulator *)
    tElapsed : TIME;  (* Elapsed cycle time *)
    bInternal : BOOL;  (* Internal work flag *)
  END_VAR
  VAR CONSTANT
    nMaxRetries : INT := 3;  (* Retry limit *)
    rScale : REAL := 1.5;  (* Setpoint scale factor *)
  END_VAR

          // 15: main state machine — 0 IDLE / 10-20 WORK / 90 DONE / 99 ERROR
CASE nState OF
    0: // IDLE — wait for enable + execute
        bBusy := FALSE;
        bDone := FALSE;
        IF bEnable AND bExecute THEN
            nState := 10;
        END_IF

    10: // WORK: acquire
        bBusy := TRUE;
        nCycleCount := nCycleCount + 1;
        fbSub(bIn := bEnable);
        nState := 20;

    20: (* WORK: process the sample and compute position *)
        rActPos := rSetpoint * rScale;
        lrAccum := lrAccum + LREAL#TO_LREAL(rActPos);
        fbTimer(bStart := TRUE, tDelay := tTimeout);
        IF fbTimer.bDone THEN
            nState := 90;
        END_IF

    90: // DONE — publish result, return to idle
        bDone := TRUE;
        bBusy := FALSE;
        nState := 0;

    99: // ERROR — latch fault
        bErr := TRUE;
        nErrId := 16#8001;
        bBusy := FALSE;
END_CASE

// Global reset path
IF bReset THEN
    bErr := FALSE;
    nErrId := 0;
    nState := 0;
END_IF
        
END_FUNCTION_BLOCK

FUNCTION_BLOCK FB_Station16
  VAR_INPUT
    bEnable : BOOL;  (* Enable this station *)
    bExecute : BOOL;  (* Trigger one work cycle *)
    bReset : BOOL;  (* Clear latched error *)
    nMode : INT := 0;  (* Operating mode selector *)
    rSetpoint : REAL := 0.0;  (* Target setpoint *)
    tTimeout : TIME := T#5S;  (* Watchdog timeout *)
    sLabel : STRING := 'station';  (* Human-readable label *)
    nStationId : DINT := 16;  (* Station identifier *)
  END_VAR
  VAR_OUTPUT
    bDone : BOOL;  (* Cycle finished *)
    bBusy : BOOL;  (* Cycle running *)
    bErr : BOOL;  (* Error latched *)
    nErrId : DINT := 0;  (* Active error code *)
    rActPos : REAL;  (* Actual position feedback *)
    nCycleCount : UDINT := 0;  (* Completed cycle counter *)
  END_VAR
  VAR
    nState : INT := 0;  (* State machine register *)
    fbSub : FB_Debounce;  (* Nested FB instance *)
    fbTimer : FB_Delay;  (* Nested FB instance *)
    anBuffer : ARRAY[0..9] OF INT;  (* Integer ring buffer *)
    arSamples : ARRAY[0..7] OF REAL;  (* Sample window *)
    lrAccum : LREAL := 0.0;  (* Long accumulator *)
    tElapsed : TIME;  (* Elapsed cycle time *)
    bInternal : BOOL;  (* Internal work flag *)
  END_VAR
  VAR CONSTANT
    nMaxRetries : INT := 3;  (* Retry limit *)
    rScale : REAL := 1.5;  (* Setpoint scale factor *)
  END_VAR

          // 16: main state machine — 0 IDLE / 10-20 WORK / 90 DONE / 99 ERROR
CASE nState OF
    0: // IDLE — wait for enable + execute
        bBusy := FALSE;
        bDone := FALSE;
        IF bEnable AND bExecute THEN
            nState := 10;
        END_IF

    10: // WORK: acquire
        bBusy := TRUE;
        nCycleCount := nCycleCount + 1;
        fbSub(bIn := bEnable);
        nState := 20;

    20: (* WORK: process the sample and compute position *)
        rActPos := rSetpoint * rScale;
        lrAccum := lrAccum + LREAL#TO_LREAL(rActPos);
        fbTimer(bStart := TRUE, tDelay := tTimeout);
        IF fbTimer.bDone THEN
            nState := 90;
        END_IF

    90: // DONE — publish result, return to idle
        bDone := TRUE;
        bBusy := FALSE;
        nState := 0;

    99: // ERROR — latch fault
        bErr := TRUE;
        nErrId := 16#8001;
        bBusy := FALSE;
END_CASE

// Global reset path
IF bReset THEN
    bErr := FALSE;
    nErrId := 0;
    nState := 0;
END_IF
        
END_FUNCTION_BLOCK

FUNCTION_BLOCK FB_Station17
  VAR_INPUT
    bEnable : BOOL;  (* Enable this station *)
    bExecute : BOOL;  (* Trigger one work cycle *)
    bReset : BOOL;  (* Clear latched error *)
    nMode : INT := 0;  (* Operating mode selector *)
    rSetpoint : REAL := 0.0;  (* Target setpoint *)
    tTimeout : TIME := T#5S;  (* Watchdog timeout *)
    sLabel : STRING := 'station';  (* Human-readable label *)
    nStationId : DINT := 17;  (* Station identifier *)
  END_VAR
  VAR_OUTPUT
    bDone : BOOL;  (* Cycle finished *)
    bBusy : BOOL;  (* Cycle running *)
    bErr : BOOL;  (* Error latched *)
    nErrId : DINT := 0;  (* Active error code *)
    rActPos : REAL;  (* Actual position feedback *)
    nCycleCount : UDINT := 0;  (* Completed cycle counter *)
  END_VAR
  VAR
    nState : INT := 0;  (* State machine register *)
    fbSub : FB_Debounce;  (* Nested FB instance *)
    fbTimer : FB_Delay;  (* Nested FB instance *)
    anBuffer : ARRAY[0..9] OF INT;  (* Integer ring buffer *)
    arSamples : ARRAY[0..7] OF REAL;  (* Sample window *)
    lrAccum : LREAL := 0.0;  (* Long accumulator *)
    tElapsed : TIME;  (* Elapsed cycle time *)
    bInternal : BOOL;  (* Internal work flag *)
  END_VAR
  VAR CONSTANT
    nMaxRetries : INT := 3;  (* Retry limit *)
    rScale : REAL := 1.5;  (* Setpoint scale factor *)
  END_VAR

          // 17: main state machine — 0 IDLE / 10-20 WORK / 90 DONE / 99 ERROR
CASE nState OF
    0: // IDLE — wait for enable + execute
        bBusy := FALSE;
        bDone := FALSE;
        IF bEnable AND bExecute THEN
            nState := 10;
        END_IF

    10: // WORK: acquire
        bBusy := TRUE;
        nCycleCount := nCycleCount + 1;
        fbSub(bIn := bEnable);
        nState := 20;

    20: (* WORK: process the sample and compute position *)
        rActPos := rSetpoint * rScale;
        lrAccum := lrAccum + LREAL#TO_LREAL(rActPos);
        fbTimer(bStart := TRUE, tDelay := tTimeout);
        IF fbTimer.bDone THEN
            nState := 90;
        END_IF

    90: // DONE — publish result, return to idle
        bDone := TRUE;
        bBusy := FALSE;
        nState := 0;

    99: // ERROR — latch fault
        bErr := TRUE;
        nErrId := 16#8001;
        bBusy := FALSE;
END_CASE

// Global reset path
IF bReset THEN
    bErr := FALSE;
    nErrId := 0;
    nState := 0;
END_IF
        
END_FUNCTION_BLOCK

FUNCTION_BLOCK FB_Station18
  VAR_INPUT
    bEnable : BOOL;  (* Enable this station *)
    bExecute : BOOL;  (* Trigger one work cycle *)
    bReset : BOOL;  (* Clear latched error *)
    nMode : INT := 0;  (* Operating mode selector *)
    rSetpoint : REAL := 0.0;  (* Target setpoint *)
    tTimeout : TIME := T#5S;  (* Watchdog timeout *)
    sLabel : STRING := 'station';  (* Human-readable label *)
    nStationId : DINT := 18;  (* Station identifier *)
  END_VAR
  VAR_OUTPUT
    bDone : BOOL;  (* Cycle finished *)
    bBusy : BOOL;  (* Cycle running *)
    bErr : BOOL;  (* Error latched *)
    nErrId : DINT := 0;  (* Active error code *)
    rActPos : REAL;  (* Actual position feedback *)
    nCycleCount : UDINT := 0;  (* Completed cycle counter *)
  END_VAR
  VAR
    nState : INT := 0;  (* State machine register *)
    fbSub : FB_Debounce;  (* Nested FB instance *)
    fbTimer : FB_Delay;  (* Nested FB instance *)
    anBuffer : ARRAY[0..9] OF INT;  (* Integer ring buffer *)
    arSamples : ARRAY[0..7] OF REAL;  (* Sample window *)
    lrAccum : LREAL := 0.0;  (* Long accumulator *)
    tElapsed : TIME;  (* Elapsed cycle time *)
    bInternal : BOOL;  (* Internal work flag *)
  END_VAR
  VAR CONSTANT
    nMaxRetries : INT := 3;  (* Retry limit *)
    rScale : REAL := 1.5;  (* Setpoint scale factor *)
  END_VAR

          // 18: main state machine — 0 IDLE / 10-20 WORK / 90 DONE / 99 ERROR
CASE nState OF
    0: // IDLE — wait for enable + execute
        bBusy := FALSE;
        bDone := FALSE;
        IF bEnable AND bExecute THEN
            nState := 10;
        END_IF

    10: // WORK: acquire
        bBusy := TRUE;
        nCycleCount := nCycleCount + 1;
        fbSub(bIn := bEnable);
        nState := 20;

    20: (* WORK: process the sample and compute position *)
        rActPos := rSetpoint * rScale;
        lrAccum := lrAccum + LREAL#TO_LREAL(rActPos);
        fbTimer(bStart := TRUE, tDelay := tTimeout);
        IF fbTimer.bDone THEN
            nState := 90;
        END_IF

    90: // DONE — publish result, return to idle
        bDone := TRUE;
        bBusy := FALSE;
        nState := 0;

    99: // ERROR — latch fault
        bErr := TRUE;
        nErrId := 16#8001;
        bBusy := FALSE;
END_CASE

// Global reset path
IF bReset THEN
    bErr := FALSE;
    nErrId := 0;
    nState := 0;
END_IF
        
END_FUNCTION_BLOCK

FUNCTION_BLOCK FB_Station19
  VAR_INPUT
    bEnable : BOOL;  (* Enable this station *)
    bExecute : BOOL;  (* Trigger one work cycle *)
    bReset : BOOL;  (* Clear latched error *)
    nMode : INT := 0;  (* Operating mode selector *)
    rSetpoint : REAL := 0.0;  (* Target setpoint *)
    tTimeout : TIME := T#5S;  (* Watchdog timeout *)
    sLabel : STRING := 'station';  (* Human-readable label *)
    nStationId : DINT := 19;  (* Station identifier *)
  END_VAR
  VAR_OUTPUT
    bDone : BOOL;  (* Cycle finished *)
    bBusy : BOOL;  (* Cycle running *)
    bErr : BOOL;  (* Error latched *)
    nErrId : DINT := 0;  (* Active error code *)
    rActPos : REAL;  (* Actual position feedback *)
    nCycleCount : UDINT := 0;  (* Completed cycle counter *)
  END_VAR
  VAR
    nState : INT := 0;  (* State machine register *)
    fbSub : FB_Debounce;  (* Nested FB instance *)
    fbTimer : FB_Delay;  (* Nested FB instance *)
    anBuffer : ARRAY[0..9] OF INT;  (* Integer ring buffer *)
    arSamples : ARRAY[0..7] OF REAL;  (* Sample window *)
    lrAccum : LREAL := 0.0;  (* Long accumulator *)
    tElapsed : TIME;  (* Elapsed cycle time *)
    bInternal : BOOL;  (* Internal work flag *)
  END_VAR
  VAR CONSTANT
    nMaxRetries : INT := 3;  (* Retry limit *)
    rScale : REAL := 1.5;  (* Setpoint scale factor *)
  END_VAR

          // 19: main state machine — 0 IDLE / 10-20 WORK / 90 DONE / 99 ERROR
CASE nState OF
    0: // IDLE — wait for enable + execute
        bBusy := FALSE;
        bDone := FALSE;
        IF bEnable AND bExecute THEN
            nState := 10;
        END_IF

    10: // WORK: acquire
        bBusy := TRUE;
        nCycleCount := nCycleCount + 1;
        fbSub(bIn := bEnable);
        nState := 20;

    20: (* WORK: process the sample and compute position *)
        rActPos := rSetpoint * rScale;
        lrAccum := lrAccum + LREAL#TO_LREAL(rActPos);
        fbTimer(bStart := TRUE, tDelay := tTimeout);
        IF fbTimer.bDone THEN
            nState := 90;
        END_IF

    90: // DONE — publish result, return to idle
        bDone := TRUE;
        bBusy := FALSE;
        nState := 0;

    99: // ERROR — latch fault
        bErr := TRUE;
        nErrId := 16#8001;
        bBusy := FALSE;
END_CASE

// Global reset path
IF bReset THEN
    bErr := FALSE;
    nErrId := 0;
    nState := 0;
END_IF
        
END_FUNCTION_BLOCK

FUNCTION_BLOCK FB_Station20
  VAR_INPUT
    bEnable : BOOL;  (* Enable this station *)
    bExecute : BOOL;  (* Trigger one work cycle *)
    bReset : BOOL;  (* Clear latched error *)
    nMode : INT := 0;  (* Operating mode selector *)
    rSetpoint : REAL := 0.0;  (* Target setpoint *)
    tTimeout : TIME := T#5S;  (* Watchdog timeout *)
    sLabel : STRING := 'station';  (* Human-readable label *)
    nStationId : DINT := 20;  (* Station identifier *)
  END_VAR
  VAR_OUTPUT
    bDone : BOOL;  (* Cycle finished *)
    bBusy : BOOL;  (* Cycle running *)
    bErr : BOOL;  (* Error latched *)
    nErrId : DINT := 0;  (* Active error code *)
    rActPos : REAL;  (* Actual position feedback *)
    nCycleCount : UDINT := 0;  (* Completed cycle counter *)
  END_VAR
  VAR
    nState : INT := 0;  (* State machine register *)
    fbSub : FB_Debounce;  (* Nested FB instance *)
    fbTimer : FB_Delay;  (* Nested FB instance *)
    anBuffer : ARRAY[0..9] OF INT;  (* Integer ring buffer *)
    arSamples : ARRAY[0..7] OF REAL;  (* Sample window *)
    lrAccum : LREAL := 0.0;  (* Long accumulator *)
    tElapsed : TIME;  (* Elapsed cycle time *)
    bInternal : BOOL;  (* Internal work flag *)
  END_VAR
  VAR CONSTANT
    nMaxRetries : INT := 3;  (* Retry limit *)
    rScale : REAL := 1.5;  (* Setpoint scale factor *)
  END_VAR

          // 20: main state machine — 0 IDLE / 10-20 WORK / 90 DONE / 99 ERROR
CASE nState OF
    0: // IDLE — wait for enable + execute
        bBusy := FALSE;
        bDone := FALSE;
        IF bEnable AND bExecute THEN
            nState := 10;
        END_IF

    10: // WORK: acquire
        bBusy := TRUE;
        nCycleCount := nCycleCount + 1;
        fbSub(bIn := bEnable);
        nState := 20;

    20: (* WORK: process the sample and compute position *)
        rActPos := rSetpoint * rScale;
        lrAccum := lrAccum + LREAL#TO_LREAL(rActPos);
        fbTimer(bStart := TRUE, tDelay := tTimeout);
        IF fbTimer.bDone THEN
            nState := 90;
        END_IF

    90: // DONE — publish result, return to idle
        bDone := TRUE;
        bBusy := FALSE;
        nState := 0;

    99: // ERROR — latch fault
        bErr := TRUE;
        nErrId := 16#8001;
        bBusy := FALSE;
END_CASE

// Global reset path
IF bReset THEN
    bErr := FALSE;
    nErrId := 0;
    nState := 0;
END_IF
        
END_FUNCTION_BLOCK

FUNCTION_BLOCK FB_Station21
  VAR_INPUT
    bEnable : BOOL;  (* Enable this station *)
    bExecute : BOOL;  (* Trigger one work cycle *)
    bReset : BOOL;  (* Clear latched error *)
    nMode : INT := 0;  (* Operating mode selector *)
    rSetpoint : REAL := 0.0;  (* Target setpoint *)
    tTimeout : TIME := T#5S;  (* Watchdog timeout *)
    sLabel : STRING := 'station';  (* Human-readable label *)
    nStationId : DINT := 21;  (* Station identifier *)
  END_VAR
  VAR_OUTPUT
    bDone : BOOL;  (* Cycle finished *)
    bBusy : BOOL;  (* Cycle running *)
    bErr : BOOL;  (* Error latched *)
    nErrId : DINT := 0;  (* Active error code *)
    rActPos : REAL;  (* Actual position feedback *)
    nCycleCount : UDINT := 0;  (* Completed cycle counter *)
  END_VAR
  VAR
    nState : INT := 0;  (* State machine register *)
    fbSub : FB_Debounce;  (* Nested FB instance *)
    fbTimer : FB_Delay;  (* Nested FB instance *)
    anBuffer : ARRAY[0..9] OF INT;  (* Integer ring buffer *)
    arSamples : ARRAY[0..7] OF REAL;  (* Sample window *)
    lrAccum : LREAL := 0.0;  (* Long accumulator *)
    tElapsed : TIME;  (* Elapsed cycle time *)
    bInternal : BOOL;  (* Internal work flag *)
  END_VAR
  VAR CONSTANT
    nMaxRetries : INT := 3;  (* Retry limit *)
    rScale : REAL := 1.5;  (* Setpoint scale factor *)
  END_VAR

          // 21: main state machine — 0 IDLE / 10-20 WORK / 90 DONE / 99 ERROR
CASE nState OF
    0: // IDLE — wait for enable + execute
        bBusy := FALSE;
        bDone := FALSE;
        IF bEnable AND bExecute THEN
            nState := 10;
        END_IF

    10: // WORK: acquire
        bBusy := TRUE;
        nCycleCount := nCycleCount + 1;
        fbSub(bIn := bEnable);
        nState := 20;

    20: (* WORK: process the sample and compute position *)
        rActPos := rSetpoint * rScale;
        lrAccum := lrAccum + LREAL#TO_LREAL(rActPos);
        fbTimer(bStart := TRUE, tDelay := tTimeout);
        IF fbTimer.bDone THEN
            nState := 90;
        END_IF

    90: // DONE — publish result, return to idle
        bDone := TRUE;
        bBusy := FALSE;
        nState := 0;

    99: // ERROR — latch fault
        bErr := TRUE;
        nErrId := 16#8001;
        bBusy := FALSE;
END_CASE

// Global reset path
IF bReset THEN
    bErr := FALSE;
    nErrId := 0;
    nState := 0;
END_IF
        
END_FUNCTION_BLOCK

FUNCTION_BLOCK FB_Station22
  VAR_INPUT
    bEnable : BOOL;  (* Enable this station *)
    bExecute : BOOL;  (* Trigger one work cycle *)
    bReset : BOOL;  (* Clear latched error *)
    nMode : INT := 0;  (* Operating mode selector *)
    rSetpoint : REAL := 0.0;  (* Target setpoint *)
    tTimeout : TIME := T#5S;  (* Watchdog timeout *)
    sLabel : STRING := 'station';  (* Human-readable label *)
    nStationId : DINT := 22;  (* Station identifier *)
  END_VAR
  VAR_OUTPUT
    bDone : BOOL;  (* Cycle finished *)
    bBusy : BOOL;  (* Cycle running *)
    bErr : BOOL;  (* Error latched *)
    nErrId : DINT := 0;  (* Active error code *)
    rActPos : REAL;  (* Actual position feedback *)
    nCycleCount : UDINT := 0;  (* Completed cycle counter *)
  END_VAR
  VAR
    nState : INT := 0;  (* State machine register *)
    fbSub : FB_Debounce;  (* Nested FB instance *)
    fbTimer : FB_Delay;  (* Nested FB instance *)
    anBuffer : ARRAY[0..9] OF INT;  (* Integer ring buffer *)
    arSamples : ARRAY[0..7] OF REAL;  (* Sample window *)
    lrAccum : LREAL := 0.0;  (* Long accumulator *)
    tElapsed : TIME;  (* Elapsed cycle time *)
    bInternal : BOOL;  (* Internal work flag *)
  END_VAR
  VAR CONSTANT
    nMaxRetries : INT := 3;  (* Retry limit *)
    rScale : REAL := 1.5;  (* Setpoint scale factor *)
  END_VAR

          // 22: main state machine — 0 IDLE / 10-20 WORK / 90 DONE / 99 ERROR
CASE nState OF
    0: // IDLE — wait for enable + execute
        bBusy := FALSE;
        bDone := FALSE;
        IF bEnable AND bExecute THEN
            nState := 10;
        END_IF

    10: // WORK: acquire
        bBusy := TRUE;
        nCycleCount := nCycleCount + 1;
        fbSub(bIn := bEnable);
        nState := 20;

    20: (* WORK: process the sample and compute position *)
        rActPos := rSetpoint * rScale;
        lrAccum := lrAccum + LREAL#TO_LREAL(rActPos);
        fbTimer(bStart := TRUE, tDelay := tTimeout);
        IF fbTimer.bDone THEN
            nState := 90;
        END_IF

    90: // DONE — publish result, return to idle
        bDone := TRUE;
        bBusy := FALSE;
        nState := 0;

    99: // ERROR — latch fault
        bErr := TRUE;
        nErrId := 16#8001;
        bBusy := FALSE;
END_CASE

// Global reset path
IF bReset THEN
    bErr := FALSE;
    nErrId := 0;
    nState := 0;
END_IF
        
END_FUNCTION_BLOCK

FUNCTION_BLOCK FB_Station23
  VAR_INPUT
    bEnable : BOOL;  (* Enable this station *)
    bExecute : BOOL;  (* Trigger one work cycle *)
    bReset : BOOL;  (* Clear latched error *)
    nMode : INT := 0;  (* Operating mode selector *)
    rSetpoint : REAL := 0.0;  (* Target setpoint *)
    tTimeout : TIME := T#5S;  (* Watchdog timeout *)
    sLabel : STRING := 'station';  (* Human-readable label *)
    nStationId : DINT := 23;  (* Station identifier *)
  END_VAR
  VAR_OUTPUT
    bDone : BOOL;  (* Cycle finished *)
    bBusy : BOOL;  (* Cycle running *)
    bErr : BOOL;  (* Error latched *)
    nErrId : DINT := 0;  (* Active error code *)
    rActPos : REAL;  (* Actual position feedback *)
    nCycleCount : UDINT := 0;  (* Completed cycle counter *)
  END_VAR
  VAR
    nState : INT := 0;  (* State machine register *)
    fbSub : FB_Debounce;  (* Nested FB instance *)
    fbTimer : FB_Delay;  (* Nested FB instance *)
    anBuffer : ARRAY[0..9] OF INT;  (* Integer ring buffer *)
    arSamples : ARRAY[0..7] OF REAL;  (* Sample window *)
    lrAccum : LREAL := 0.0;  (* Long accumulator *)
    tElapsed : TIME;  (* Elapsed cycle time *)
    bInternal : BOOL;  (* Internal work flag *)
  END_VAR
  VAR CONSTANT
    nMaxRetries : INT := 3;  (* Retry limit *)
    rScale : REAL := 1.5;  (* Setpoint scale factor *)
  END_VAR

          // 23: main state machine — 0 IDLE / 10-20 WORK / 90 DONE / 99 ERROR
CASE nState OF
    0: // IDLE — wait for enable + execute
        bBusy := FALSE;
        bDone := FALSE;
        IF bEnable AND bExecute THEN
            nState := 10;
        END_IF

    10: // WORK: acquire
        bBusy := TRUE;
        nCycleCount := nCycleCount + 1;
        fbSub(bIn := bEnable);
        nState := 20;

    20: (* WORK: process the sample and compute position *)
        rActPos := rSetpoint * rScale;
        lrAccum := lrAccum + LREAL#TO_LREAL(rActPos);
        fbTimer(bStart := TRUE, tDelay := tTimeout);
        IF fbTimer.bDone THEN
            nState := 90;
        END_IF

    90: // DONE — publish result, return to idle
        bDone := TRUE;
        bBusy := FALSE;
        nState := 0;

    99: // ERROR — latch fault
        bErr := TRUE;
        nErrId := 16#8001;
        bBusy := FALSE;
END_CASE

// Global reset path
IF bReset THEN
    bErr := FALSE;
    nErrId := 0;
    nState := 0;
END_IF
        
END_FUNCTION_BLOCK

FUNCTION_BLOCK FB_Station24
  VAR_INPUT
    bEnable : BOOL;  (* Enable this station *)
    bExecute : BOOL;  (* Trigger one work cycle *)
    bReset : BOOL;  (* Clear latched error *)
    nMode : INT := 0;  (* Operating mode selector *)
    rSetpoint : REAL := 0.0;  (* Target setpoint *)
    tTimeout : TIME := T#5S;  (* Watchdog timeout *)
    sLabel : STRING := 'station';  (* Human-readable label *)
    nStationId : DINT := 24;  (* Station identifier *)
  END_VAR
  VAR_OUTPUT
    bDone : BOOL;  (* Cycle finished *)
    bBusy : BOOL;  (* Cycle running *)
    bErr : BOOL;  (* Error latched *)
    nErrId : DINT := 0;  (* Active error code *)
    rActPos : REAL;  (* Actual position feedback *)
    nCycleCount : UDINT := 0;  (* Completed cycle counter *)
  END_VAR
  VAR
    nState : INT := 0;  (* State machine register *)
    fbSub : FB_Debounce;  (* Nested FB instance *)
    fbTimer : FB_Delay;  (* Nested FB instance *)
    anBuffer : ARRAY[0..9] OF INT;  (* Integer ring buffer *)
    arSamples : ARRAY[0..7] OF REAL;  (* Sample window *)
    lrAccum : LREAL := 0.0;  (* Long accumulator *)
    tElapsed : TIME;  (* Elapsed cycle time *)
    bInternal : BOOL;  (* Internal work flag *)
  END_VAR
  VAR CONSTANT
    nMaxRetries : INT := 3;  (* Retry limit *)
    rScale : REAL := 1.5;  (* Setpoint scale factor *)
  END_VAR

          // 24: main state machine — 0 IDLE / 10-20 WORK / 90 DONE / 99 ERROR
CASE nState OF
    0: // IDLE — wait for enable + execute
        bBusy := FALSE;
        bDone := FALSE;
        IF bEnable AND bExecute THEN
            nState := 10;
        END_IF

    10: // WORK: acquire
        bBusy := TRUE;
        nCycleCount := nCycleCount + 1;
        fbSub(bIn := bEnable);
        nState := 20;

    20: (* WORK: process the sample and compute position *)
        rActPos := rSetpoint * rScale;
        lrAccum := lrAccum + LREAL#TO_LREAL(rActPos);
        fbTimer(bStart := TRUE, tDelay := tTimeout);
        IF fbTimer.bDone THEN
            nState := 90;
        END_IF

    90: // DONE — publish result, return to idle
        bDone := TRUE;
        bBusy := FALSE;
        nState := 0;

    99: // ERROR — latch fault
        bErr := TRUE;
        nErrId := 16#8001;
        bBusy := FALSE;
END_CASE

// Global reset path
IF bReset THEN
    bErr := FALSE;
    nErrId := 0;
    nState := 0;
END_IF
        
END_FUNCTION_BLOCK

FUNCTION F_ClampReal : REAL
  VAR_INPUT
    rValue : REAL;  (* Value to clamp *)
    rMin : REAL;  (* Lower bound *)
    rMax : REAL;  (* Upper bound *)
  END_VAR

          IF rValue < rMin THEN
    F_ClampReal := rMin;
ELSIF rValue > rMax THEN
    F_ClampReal := rMax;
ELSE
    F_ClampReal := rValue;
END_IF
        
END_FUNCTION

FUNCTION F_ScaleInt : DINT
  VAR_INPUT
    nRaw : INT;  (* Raw reading *)
    nFactor : DINT;  (* Scale factor *)
  END_VAR

          F_ScaleInt := DINT#TO_DINT(nRaw) * nFactor;
        
END_FUNCTION

PROGRAM PRG_Main
  VAR
    fbStation01 : FB_Station01;  (* Station 01 instance *)
    fbStation02 : FB_Station02;  (* Station 02 instance *)
    fbStation03 : FB_Station03;  (* Station 03 instance *)
    fbStation04 : FB_Station04;  (* Station 04 instance *)
    fbStation05 : FB_Station05;  (* Station 05 instance *)
    fbStation06 : FB_Station06;  (* Station 06 instance *)
    fbStation07 : FB_Station07;  (* Station 07 instance *)
    fbStation08 : FB_Station08;  (* Station 08 instance *)
    fbStation09 : FB_Station09;  (* Station 09 instance *)
    fbStation10 : FB_Station10;  (* Station 10 instance *)
    fbStation11 : FB_Station11;  (* Station 11 instance *)
    fbStation12 : FB_Station12;  (* Station 12 instance *)
    fbStation13 : FB_Station13;  (* Station 13 instance *)
    fbStation14 : FB_Station14;  (* Station 14 instance *)
    fbStation15 : FB_Station15;  (* Station 15 instance *)
    fbStation16 : FB_Station16;  (* Station 16 instance *)
    fbStation17 : FB_Station17;  (* Station 17 instance *)
    fbStation18 : FB_Station18;  (* Station 18 instance *)
    fbStation19 : FB_Station19;  (* Station 19 instance *)
    fbStation20 : FB_Station20;  (* Station 20 instance *)
    fbStation21 : FB_Station21;  (* Station 21 instance *)
    fbStation22 : FB_Station22;  (* Station 22 instance *)
    fbStation23 : FB_Station23;  (* Station 23 instance *)
    fbStation24 : FB_Station24;  (* Station 24 instance *)
    nHeartbeat : UDINT := 0;  (* Free-running heartbeat *)
    bTick : BOOL;  (* One-shot execute pulse *)
    bClearAll : BOOL;  (* Broadcast reset *)
    rLineSpeed : REAL := 0.0;  (* Current line speed *)
    tScanTime : TIME;  (* Measured scan time *)
    sStatus : STRING := 'RUN';  (* Status text *)
  END_VAR

          // Heartbeat + broadcast drive of all stations
nHeartbeat := nHeartbeat + 1;

fbStation01(bEnable := GVL_Machine.bMachineReady, bExecute := bTick, bReset := bClearAll);
fbStation02(bEnable := GVL_Machine.bMachineReady, bExecute := bTick, bReset := bClearAll);
fbStation03(bEnable := GVL_Machine.bMachineReady, bExecute := bTick, bReset := bClearAll);
fbStation04(bEnable := GVL_Machine.bMachineReady, bExecute := bTick, bReset := bClearAll);
fbStation05(bEnable := GVL_Machine.bMachineReady, bExecute := bTick, bReset := bClearAll);
fbStation06(bEnable := GVL_Machine.bMachineReady, bExecute := bTick, bReset := bClearAll);
fbStation07(bEnable := GVL_Machine.bMachineReady, bExecute := bTick, bReset := bClearAll);
fbStation08(bEnable := GVL_Machine.bMachineReady, bExecute := bTick, bReset := bClearAll);
fbStation09(bEnable := GVL_Machine.bMachineReady, bExecute := bTick, bReset := bClearAll);
fbStation10(bEnable := GVL_Machine.bMachineReady, bExecute := bTick, bReset := bClearAll);
fbStation11(bEnable := GVL_Machine.bMachineReady, bExecute := bTick, bReset := bClearAll);
fbStation12(bEnable := GVL_Machine.bMachineReady, bExecute := bTick, bReset := bClearAll);
fbStation13(bEnable := GVL_Machine.bMachineReady, bExecute := bTick, bReset := bClearAll);
fbStation14(bEnable := GVL_Machine.bMachineReady, bExecute := bTick, bReset := bClearAll);
fbStation15(bEnable := GVL_Machine.bMachineReady, bExecute := bTick, bReset := bClearAll);
fbStation16(bEnable := GVL_Machine.bMachineReady, bExecute := bTick, bReset := bClearAll);
fbStation17(bEnable := GVL_Machine.bMachineReady, bExecute := bTick, bReset := bClearAll);
fbStation18(bEnable := GVL_Machine.bMachineReady, bExecute := bTick, bReset := bClearAll);
fbStation19(bEnable := GVL_Machine.bMachineReady, bExecute := bTick, bReset := bClearAll);
fbStation20(bEnable := GVL_Machine.bMachineReady, bExecute := bTick, bReset := bClearAll);
fbStation21(bEnable := GVL_Machine.bMachineReady, bExecute := bTick, bReset := bClearAll);
fbStation22(bEnable := GVL_Machine.bMachineReady, bExecute := bTick, bReset := bClearAll);
fbStation23(bEnable := GVL_Machine.bMachineReady, bExecute := bTick, bReset := bClearAll);
fbStation24(bEnable := GVL_Machine.bMachineReady, bExecute := bTick, bReset := bClearAll);

IF GVL_Machine.nActiveStation > GVL_Config.nMaxStations THEN
    bClearAll := TRUE;
END_IF
        
END_PROGRAM
